FUNCTION_BLOCK Q_NumericValue_PHYSA_LREAL (* Command change numeric value — accepts physical LREAL value via ALR adapter (wraps Q_NumericValue_PHYS_LREAL) *)
  (* Standard: ISO 11783-6; Description: Copyright (c) 2026 Meisterschulen am Ostbahnhof This program and the accompanying materials are made available under the terms of the Eclipse Public License 2.0 which is available at https://www.eclipse.org/legal/epl-2.0/ SPDX-License-Identifier: EPL-2.0 *)
  (* Version 1.0, 2026-04-21, Franz Höpfinger, Meisterschulen am Ostbahnhof, initial API and implementation *)
  PACKAGE isobus::UT::Q;
  IMPORT isobus::UT::Q::const::IDs::ID_NULL;
  IMPORT logiBUS::utils::conversion::phys::NumericObjectPool_S;
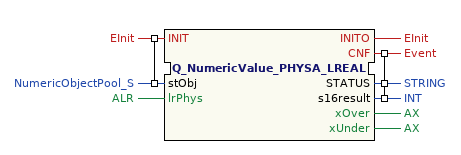
  EVENT_INPUT
    INIT : EInit WITH stObj; (* Service Initialization *)
  END_EVENT
  EVENT_OUTPUT
    INITO : EInit; (* Initialization Confirm *)
    CNF WITH STATUS, s16result; (* Confirmation of Requested Service *)
  END_EVENT
  VAR_INPUT
    stObj : logiBUS::utils::conversion::phys::NumericObjectPool_S := (u16ObjId := ID_NULL, r32Scale := 1.0, i32Offset := 0, u8Decimals := 0); (* Object pool properties (u16ObjId, scale, offset, decimals) *)
  END_VAR
  VAR_OUTPUT
    STATUS : STRING; (* Service Status *)
    s16result : INT; (* retval see Q_NumericValue *)
  END_VAR
  SOCKETS
    lrPhys : adapter::types::unidirectional::ALR; (* Physical LREAL value input *)
  END_SOCKETS
  PLUGS
    xOver : adapter::types::unidirectional::AX; (* Physical value exceeds upper ISOBUS limit *)
    xUnder : adapter::types::unidirectional::AX; (* Physical value below lower ISOBUS limit *)
  END_PLUGS
  FBS
    Q_NumericValue_PHYS_LREAL : isobus::UT::Q::Q_NumericValue_PHYS_LREAL;
  END_FBS
  EVENT_CONNECTIONS
    INIT TO Q_NumericValue_PHYS_LREAL.INIT;
    lrPhys.E1 TO Q_NumericValue_PHYS_LREAL.REQ;
    Q_NumericValue_PHYS_LREAL.INITO TO INITO;
    Q_NumericValue_PHYS_LREAL.CNF TO CNF;
    Q_NumericValue_PHYS_LREAL.CNF TO xUnder.E1;
    Q_NumericValue_PHYS_LREAL.CNF TO xOver.E1;
  END_CONNECTIONS
  DATA_CONNECTIONS
    stObj TO Q_NumericValue_PHYS_LREAL.stObj;
    lrPhys.D1 TO Q_NumericValue_PHYS_LREAL.lrPhys;
    Q_NumericValue_PHYS_LREAL.STATUS TO STATUS;
    Q_NumericValue_PHYS_LREAL.s16result TO s16result;
    Q_NumericValue_PHYS_LREAL.xOver TO xOver.D1;
    Q_NumericValue_PHYS_LREAL.xUnder TO xUnder.D1;
  END_CONNECTIONS
END_FUNCTION_BLOCK
